Fanuc KAREL source: NC0046.KL

-- PROVISIONAL review KL for V770-1; original PC SHA256 4277b0ae20a96910ea56f7f9a0cc738120b6ebd74a6a18a9e79206c1668f23d3
-- Incomplete behavior may be omitted. Consult companion uncertainty JSON. Do not deploy.
PROGRAM NC0046
%NOLOCKGROUP
-- UNRESOLVED_LOCAL_POOL 1 cells at code offset 3; source declarations unknown
-- DIRECT_LOCAL_WORD_ACCESS alone does not prove INTEGER, REAL, or BOOLEAN
BEGIN
  -- UNRESOLVED_PC offsets 0-8; opcodes 2B,2C,7B
  -- UNRESOLVED_PC offsets 13-20; opcodes 9D,23
  -- UNRESOLVED_PC offsets 25-38; opcodes 21,9D,57,79
  -- UNRESOLVED_PC offsets 43-60; opcodes 21,40,41,42
  -- UNRESOLVED_PC offsets 65-78; opcodes 21,9D,57,79
  -- UNRESOLVED_PC offsets 83-100; opcodes 21,40,41,42
  -- UNRESOLVED_PC offsets 105-118; opcodes 21,9D,57,79
  -- UNRESOLVED_PC offsets 123-140; opcodes 21,40,41,42
  -- UNRESOLVED_PC offsets 145-158; opcodes 21,9D,57,79
  -- UNRESOLVED_PC offsets 163-180; opcodes 21,40,41,42
  -- UNRESOLVED_PC offsets 185-215; opcodes 21,9D,52,23,7A,40,41,42
  -- UNRESOLVED_PC offsets 220-244; opcodes 21,2E,52,23,7A,43
  -- UNRESOLVED_PC offsets 249-267; opcodes 21,2E,52,23
  -- UNRESOLVED_PC offsets 277-282; opcodes 7A
  -- UNRESOLVED_PC offsets 287-305; opcodes 21,2E,52,23
  -- UNRESOLVED_PC offsets 310-326; opcodes 7A,40,41,42
  -- UNRESOLVED_PC offsets 331-355; opcodes 21,2E,52,23,7A,43
  -- UNRESOLVED_PC offsets 360-378; opcodes 21,2E,52,23
  -- UNRESOLVED_PC offsets 388-393; opcodes 7A
  -- UNRESOLVED_PC offsets 398-416; opcodes 21,2E,52,23
  -- UNRESOLVED_PC offsets 421-437; opcodes 7A,40,41,42
  -- UNRESOLVED_PC offsets 442-466; opcodes 21,2E,52,23,7A,43
  -- UNRESOLVED_PC offsets 471-489; opcodes 21,2E,52,23
  -- UNRESOLVED_PC offsets 499-504; opcodes 7A
  -- UNRESOLVED_PC offsets 509-527; opcodes 21,2E,52,23
  -- UNRESOLVED_PC offsets 532-548; opcodes 7A,40,41,42
  -- UNRESOLVED_PC offsets 553-577; opcodes 21,2E,52,23,7A,43
  -- UNRESOLVED_PC offsets 582-600; opcodes 21,2E,52,23
  -- UNRESOLVED_PC offsets 610-615; opcodes 7A
  -- UNRESOLVED_PC offsets 620-638; opcodes 21,2E,52,23
  -- UNRESOLVED_PC offsets 648-652; opcodes 7F
  -- UNRESOLVED_PC offsets 657-661; opcodes 27,AA
  -- UNRESOLVED_PC offsets 666-670; opcodes 7F
END NC0046
